# EPICS autosave request: gardasoftLED/RTSeriesChannel_settings.req
$(P):CH$(N):ON
$(P):CH$(N):OPTIONS:SET-01
$(P):CH$(N):OPTIONS:SET-02
$(P):CH$(N):OPTIONS:SET-03
$(P):CH$(N):OPTIONS:SET-06
$(P):CH$(N):SETMAXCURRENT
$(P):CH$(N):SETMAXVOLTAGE
$(P):CH$(N):SETOPTIONS
$(P):CH$(N):SETOUTPUT
